ADAPTER EVENT_HS_ACK_WSTRING (* Handshake family, request/confirm with WSTRING payload: CNF/CNFD in, REQ/REQD out, no IND/RSP *)
  (* Standard: 61499-1; Description: Copyright (c) 2026 HR Agrartechnik GmbH This program and the accompanying materials are made available under the terms of the Eclipse Public License 2.0 which is available at https://www.eclipse.org/legal/epl-2.0/ SPDX-License-Identifier: EPL-2.0 *)
  (* Version 1.0, 2026-09-02, Franz Höpfinger, HR Agrartechnik GmbH, Data-carrying variant of EVENT_HS_ACK: adds WSTRING payloads (REQD/CNFD) to the request/confirm pair, matching the 'name,value' message style (e.g. push,100) documented in HandshakePattern.md *)
  PACKAGE adapter::types::bidirectional::Handshake;
  (* Documentation:
  Data-carrying variant of EVENT_HS_ACK (reduced member of the EVENT_HS family, Handshake design pattern, IEC 61499 primer course, Module 6, Valeriy Vyatkin), keeping only the request/confirm half of the full REQ/CNF/IND/RSP vocabulary, each with a WSTRING payload:
    - REQ / REQD – request + payload, from Plug to Socket (e.g. "push,100")
   - CNF / CNFD – confirmation + payload, from Socket to Plug, answers a REQ (e.g. "push,100")
    No IND/RSP (and no INDD/RSPD): the Socket side can only ever answer a REQ with a CNF, it can never push an unsolicited indication back to the Plug.
   Same Socket/Plug role split as EVENT_HS: Plug (Name>>) keeps the declared direction and plays the Requester/client role: it fires REQ/REQD and reacts to CNF/CNFD. Socket (>>Name) mirrors the direction and plays the Responder/server role: it reacts to REQ/REQD and fires CNF/CNFD.
   See test_AX/Meins/DesingPatterns/HandshakePattern/HandshakePattern.md for the full write-up of the EVENT_HS family, including this and the other three reduced variants (EVENT_HS_UNI, EVENT_HS_UNI_WSTRING, EVENT_HS_ACK).
  *)
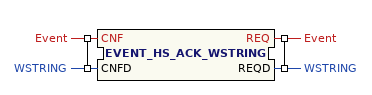
  EVENT_INPUT
    CNF WITH CNFD; (* Confirmation from Socket to Plug, answers a REQ *)
  END_EVENT
  EVENT_OUTPUT
    REQ WITH REQD; (* Request from Plug to Socket *)
  END_EVENT
  VAR_INPUT
    CNFD : WSTRING; (* Confirmation payload, accompanies CNF *)
  END_VAR
  VAR_OUTPUT
    REQD : WSTRING; (* Request payload, accompanies REQ *)
  END_VAR
  SERVICE PLUG/SOCKET
    SEQUENCE request_confirm
      PLUG.REQ(REQD) -> SOCKET.REQ(REQD);
      SOCKET.CNF(CNFD) -> PLUG.CNF(CNFD);
    END_SEQUENCE
  END_SERVICE
END_ADAPTER
